# EPICS autosave request: throttleApp/Db/throttle.req
$(P)$(THR).PREC
$(P)$(THR).DPREC
$(P)$(THR).OUT
$(P)$(THR).DLY
